// TIA Portal V18 export
FUNCTION_BLOCK "Analog_Valve"   // FB104, FBD
TITLE = Analog Valve Control
{ S7_Optimized_Access := 'FALSE' }
AUTHOR : THE
FAMILY : MAIN
NAME : PVALVE
VERSION : 1.1
// stored: AutoNumber false, IsIECCheckEnabled false, SetENOAutomatically false, UDAEnableTagReadback false
   VAR_INPUT
      IN_Em_Stop : Bool;   // Emergency stop / 1=OK, 0=Not OK
      IN_Interlock : Bool;   // Interlock when valve in auto mode / 0=OK, 1=Interlocked
      IN_Reset : Bool;   // Reset alarm / Cmd: Reset
      IN_ValveSP : Real;   // Cmd: Setpoint 0-100%
      IN_ValveSP_Min : Real;   // Min value of the Input Setpoint
      IN_ValveSP_Max : Real;   // Max value of the Iinput setpoint
      IN_Valve_Feedback : Real;   // Sts: Valve feedback 0-100%
      IN_TimerSetpointNotReached : Timer;   // Open % / Close time for valve (sec) / Timer number Setpoint Not Reached
      IN_TimerNotClosing : Timer;   // Timer number Not closing
      IN_TimeoutTime1 : S5Time;   // Real Feedback from Valve / Timeout time in Sec
      IN_TimeoutTime2 : S5Time;   // Timeout time in Sec
   END_VAR
   VAR_OUTPUT
      OUT_ValveSP : Real;   // Setpoint 0-100% Output
      OUT_Valve_Feedback : Real;   // Sts_Valve Feedback 0-100%
      OUT_Valve_Closed : Bool;   // Status: Valve Closed / Sts: Valve closed 1=Closed,0=open
      OUT_Valve_Not_Closing : Bool;   // Alarm: valve not closing / Sts: Timeout Valve Closing
      OUT_SP_Not_Reached : Bool;   // Sts: Setpoint not Reached
      OUT_ValveSP_OOR : Bool;   // Setpoint Value Out Of Range
   END_VAR
   VAR DB_SPECIFIC
      Valve_SP : Real;
      Pos_Deviation_Valve : Real;
      Neg_Deviation_Valve : Real;
      Open_Cmd : Bool;
      Operate : Bool;
   END_VAR
   VAR_TEMP
      SP_Overrange : Bool;
      SP_Underrange : Bool;
   END_VAR
   VAR_TEMP   // added for the SCL form of the ladder/FBD networks
      _w1 : Bool;
      _s5time1 : S5Time;
   END_VAR
BEGIN

REGION Network 1: Internal operate flag
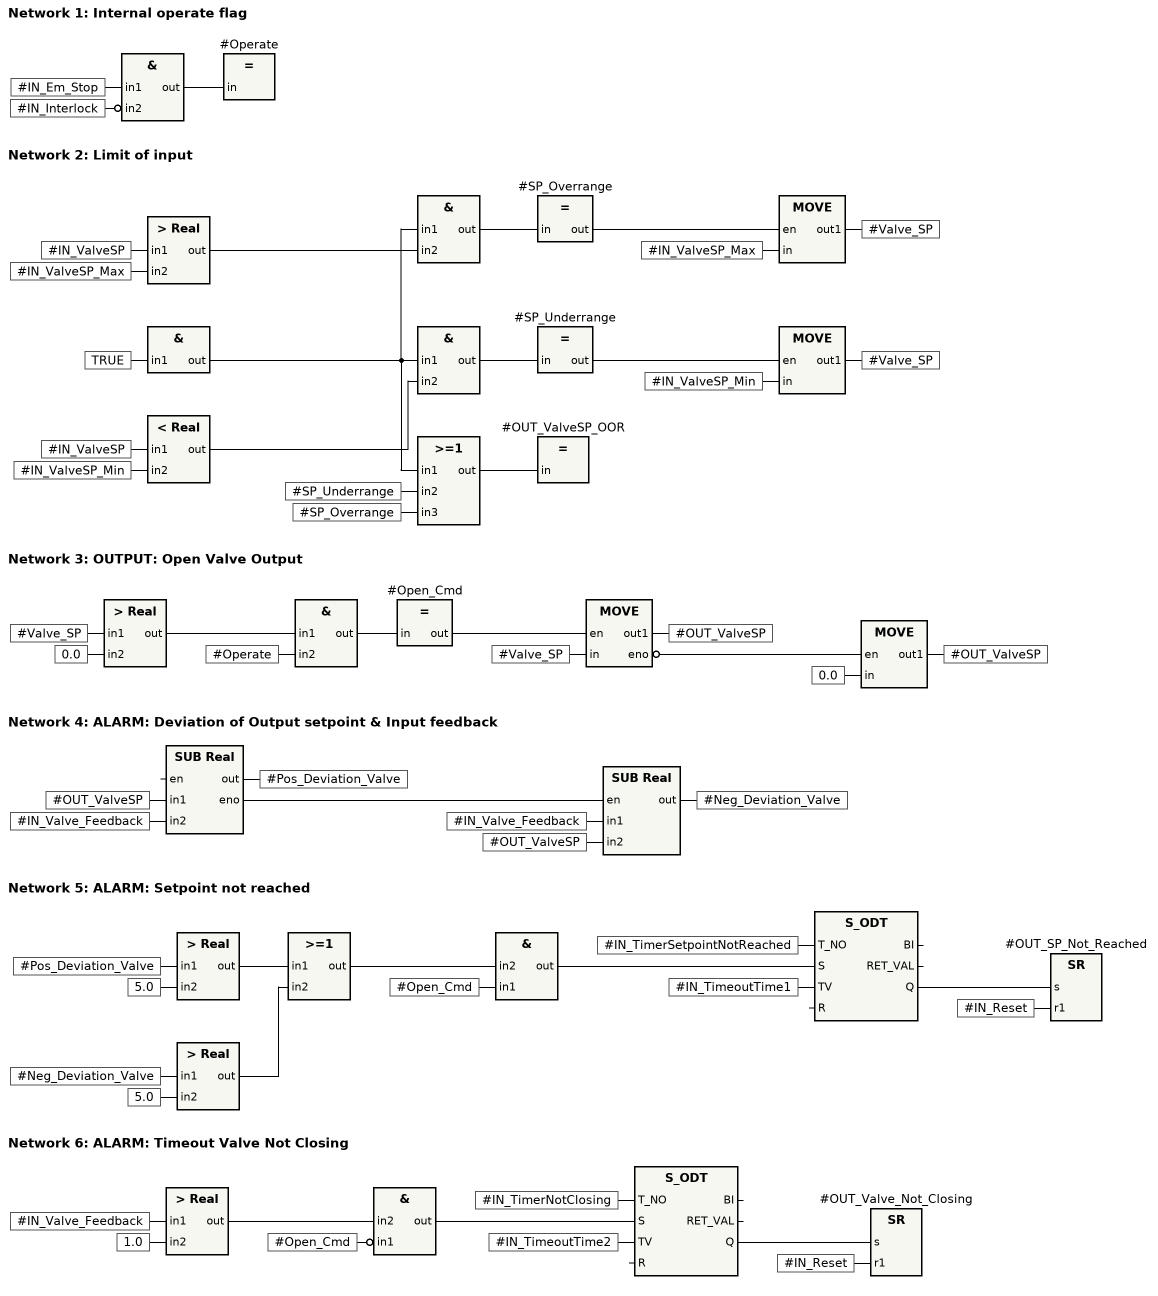
   #Operate := #IN_Em_Stop AND NOT #IN_Interlock;
END_REGION

REGION Network 2: Limit of input
   #SP_Overrange := TRUE AND (#IN_ValveSP > #IN_ValveSP_Max);
   IF #SP_Overrange THEN #Valve_SP := #IN_ValveSP_Max; END_IF;
   #SP_Underrange := TRUE AND (#IN_ValveSP < #IN_ValveSP_Min);
   IF #SP_Underrange THEN #Valve_SP := #IN_ValveSP_Min; END_IF;
   #OUT_ValveSP_OOR := TRUE OR #SP_Underrange OR #SP_Overrange;
END_REGION

REGION Network 3: OUTPUT: Open Valve Output
   #Open_Cmd := (#Valve_SP > 0.0) AND #Operate;
   IF #Open_Cmd THEN #OUT_ValveSP := #Valve_SP; END_IF;
   IF NOT #Open_Cmd THEN #OUT_ValveSP := 0.0; END_IF;
END_REGION

REGION Network 4: ALARM: Deviation of Output setpoint & Input feedback
   // Check if deviation between Output & Fedback
   // ENO of a box is taken as its EN; it also drops when the box reports an error
   #Pos_Deviation_Valve := #OUT_ValveSP - #IN_Valve_Feedback;
   #Neg_Deviation_Valve := #IN_Valve_Feedback - #OUT_ValveSP;
END_REGION

REGION Network 5: ALARM: Setpoint not reached
   #_s5time1 := S_ODT(T_NO := #IN_TimerSetpointNotReached,
                      S := ((#Pos_Deviation_Valve > 5.0) OR (#Neg_Deviation_Valve > 5.0)) AND #Open_Cmd,
                      TV := #IN_TimeoutTime1,
                      Q => #_w1);
   IF #_w1 THEN
       #OUT_SP_Not_Reached := TRUE;   // SR flip-flop
   END_IF;
   IF #IN_Reset THEN #OUT_SP_Not_Reached := FALSE; END_IF;
END_REGION

REGION Network 6: ALARM: Timeout Valve Not Closing
   #_s5time1 := S_ODT(T_NO := #IN_TimerNotClosing,
                      S := (#IN_Valve_Feedback > 1.0) AND NOT #Open_Cmd,
                      TV := #IN_TimeoutTime2,
                      Q => #_w1);
   IF #_w1 THEN
       #OUT_Valve_Not_Closing := TRUE;   // SR flip-flop
   END_IF;
   IF #IN_Reset THEN #OUT_Valve_Not_Closing := FALSE; END_IF;
END_REGION

REGION Network 7: OUTPUT: Valve Feedback to Output
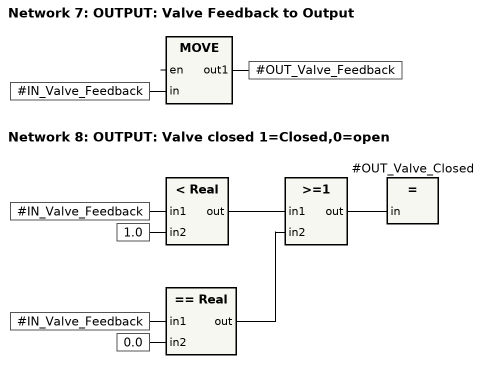
   #OUT_Valve_Feedback := #IN_Valve_Feedback;
END_REGION

REGION Network 8: OUTPUT: Valve closed 1=Closed,0=open
   #OUT_Valve_Closed := (#IN_Valve_Feedback < 1.0) OR (#IN_Valve_Feedback = 0.0);
END_REGION
END_FUNCTION_BLOCK
